FUNCTION_BLOCK L3_OrderManager (* Composite Function Block Type *)
  (* Standard: 61499-2 *)
  (* Version 0.0, 2014-10-02, EQUEROL, UJI *)
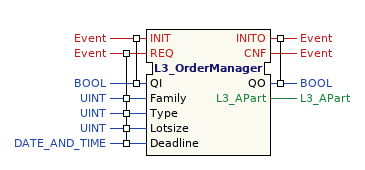
  EVENT_INPUT
    INIT WITH QI; (* Initialization Request *)
    REQ WITH Family, Type, Lotsize, Deadline; (* Normal Execution Request *)
  END_EVENT
  EVENT_OUTPUT
    INITO WITH QO; (* Initialization Confirm *)
    CNF; (* Execution Confirmation *)
  END_EVENT
  VAR_INPUT
    QI : BOOL; (* Input event qualifier *)
    Family : UINT; (* Family od the parts to be manufactured *)
    Type : UINT; (* Type of the parts to be manufactured *)
    Lotsize : UINT; (* Number of part to be manufactured *)
    Deadline : DATE_AND_TIME; (* Order delivery date and time *)
  END_VAR
  VAR_OUTPUT
    QO : BOOL; (* Output event qualifier *)
  END_VAR
  PLUGS
    L3_APart : L3_APart;
  END_PLUGS
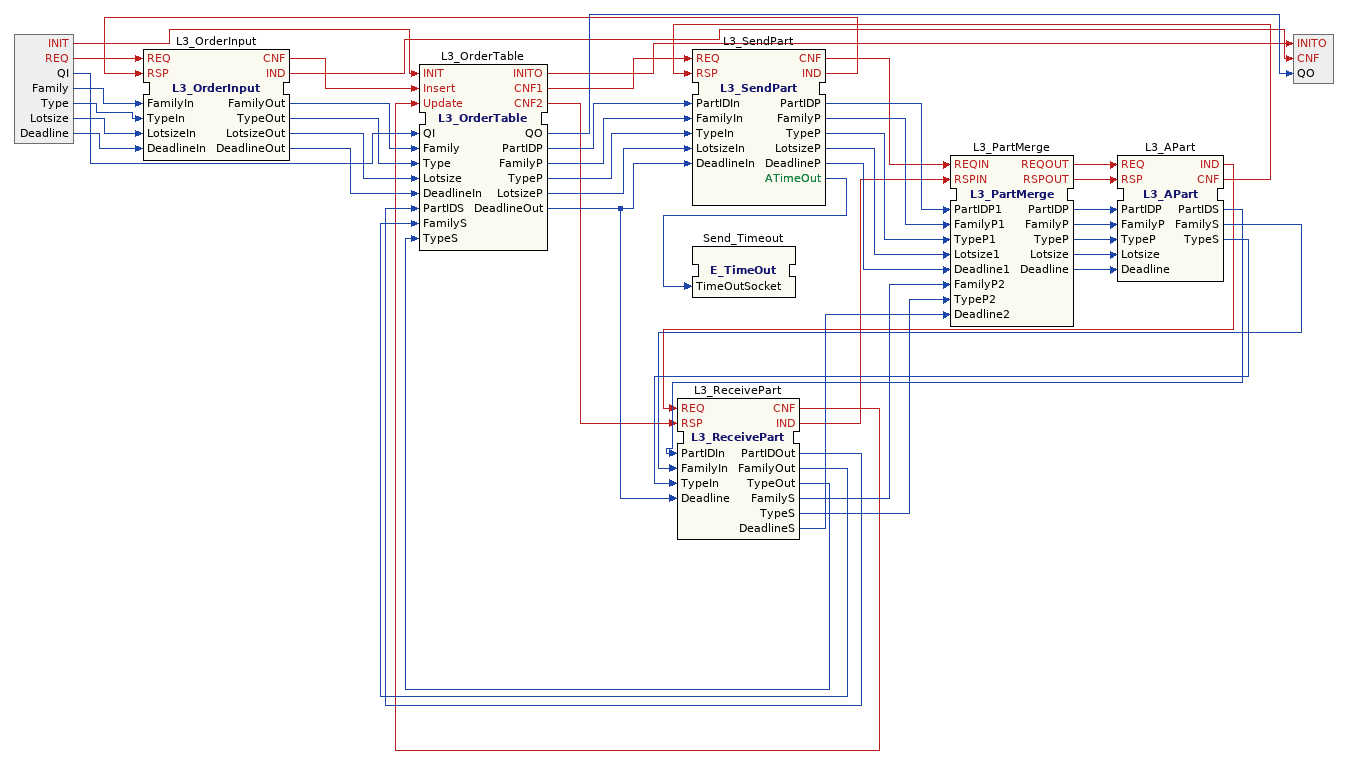
  FBS
    L3_OrderTable : L3_OrderTable;
    L3_ReceivePart : L3_ReceivePart;
    L3_SendPart : L3_SendPart;
    Send_Timeout : E_TimeOut;
    L3_OrderInput : L3_OrderInput;
    L3_PartMerge : L3_PartMerge;
  END_FBS
  EVENT_CONNECTIONS
    L3_OrderTable.CNF1 TO L3_SendPart.REQ;
    L3_ReceivePart.CNF TO L3_OrderTable.Update;
    L3_OrderTable.CNF2 TO L3_ReceivePart.RSP;
    L3_OrderInput.CNF TO L3_OrderTable.Insert;
    L3_SendPart.IND TO L3_OrderInput.RSP;
    L3_APart.IND TO L3_ReceivePart.REQ;
    L3_APart.CNF TO L3_SendPart.RSP;
    L3_SendPart.CNF TO L3_PartMerge.REQIN;
    L3_ReceivePart.IND TO L3_PartMerge.RSPIN;
    L3_PartMerge.REQOUT TO L3_APart.REQ;
    L3_PartMerge.RSPOUT TO L3_APart.RSP;
    REQ TO L3_OrderInput.REQ;
    INIT TO L3_OrderTable.INIT;
    L3_OrderTable.INITO TO INITO;
    L3_OrderInput.IND TO CNF;
  END_CONNECTIONS
  DATA_CONNECTIONS
    L3_OrderTable.PartIDP TO L3_SendPart.PartIDIn;
    L3_OrderTable.FamilyP TO L3_SendPart.FamilyIn;
    L3_OrderTable.TypeP TO L3_SendPart.TypeIn;
    L3_OrderTable.LotsizeP TO L3_SendPart.LotsizeIn;
    L3_OrderTable.DeadlineOut TO L3_SendPart.DeadlineIn;
    L3_SendPart.ATimeOut TO Send_Timeout.TimeOutSocket;
    L3_ReceivePart.PartIDOut TO L3_OrderTable.PartIDS;
    L3_ReceivePart.FamilyOut TO L3_OrderTable.FamilyS;
    L3_ReceivePart.TypeOut TO L3_OrderTable.TypeS;
    L3_OrderTable.DeadlineOut TO L3_ReceivePart.Deadline;
    L3_OrderInput.FamilyOut TO L3_OrderTable.Family;
    L3_OrderInput.TypeOut TO L3_OrderTable.Type;
    L3_OrderInput.LotsizeOut TO L3_OrderTable.Lotsize;
    L3_OrderInput.DeadlineOut TO L3_OrderTable.DeadlineIn;
    L3_APart.PartIDS TO L3_ReceivePart.PartIDIn;
    L3_APart.FamilyS TO L3_ReceivePart.FamilyIn;
    L3_APart.TypeS TO L3_ReceivePart.TypeIn;
    L3_SendPart.PartIDP TO L3_PartMerge.PartIDP1;
    L3_SendPart.FamilyP TO L3_PartMerge.FamilyP1;
    L3_SendPart.TypeP TO L3_PartMerge.TypeP1;
    L3_SendPart.LotsizeP TO L3_PartMerge.Lotsize1;
    L3_SendPart.DeadlineP TO L3_PartMerge.Deadline1;
    L3_ReceivePart.FamilyS TO L3_PartMerge.FamilyP2;
    L3_ReceivePart.TypeS TO L3_PartMerge.TypeP2;
    L3_ReceivePart.DeadlineS TO L3_PartMerge.Deadline2;
    L3_PartMerge.PartIDP TO L3_APart.PartIDP;
    L3_PartMerge.FamilyP TO L3_APart.FamilyP;
    L3_PartMerge.TypeP TO L3_APart.TypeP;
    L3_PartMerge.Lotsize TO L3_APart.Lotsize;
    L3_PartMerge.Deadline TO L3_APart.Deadline;
    Family TO L3_OrderInput.FamilyIn;
    Type TO L3_OrderInput.TypeIn;
    Lotsize TO L3_OrderInput.LotsizeIn;
    Deadline TO L3_OrderInput.DeadlineIn;
    QI TO L3_OrderTable.QI;
    L3_OrderTable.QO TO QO;
  END_CONNECTIONS
END_FUNCTION_BLOCK
